TYPE DCTIME64_UINT :
STRUCT
	tDC : T_DCTIME64;
	iData : UINT;
END_STRUCT
END_TYPE

(* stored: Version 1.1.0.1, ProductVersion 3.1.4022.10
   DUT DCTIME64_UINT: Id {dc470cd3-fa53-42f6-88b6-afc6281bf163} *)
